Yaskawa INFORM job: FACE.JBI

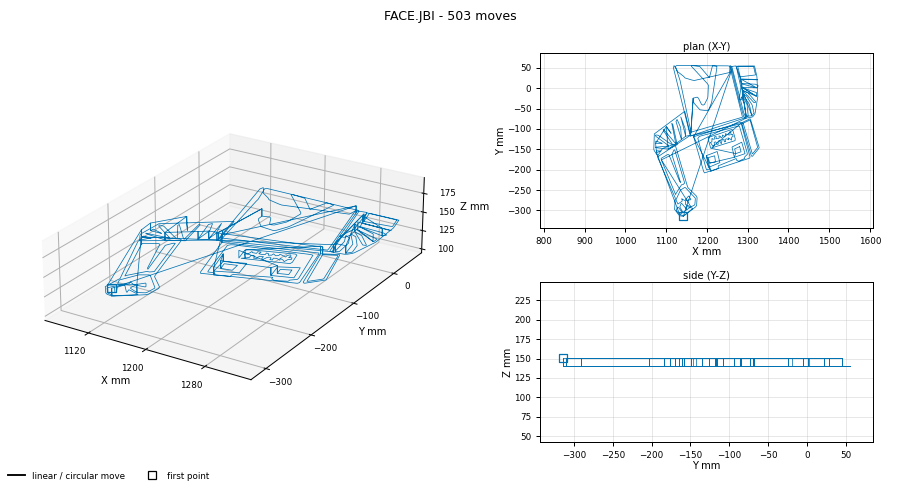
[picture p0: tool path of FACE.JBI, 503 of 503 moves have a stored position in this frame; points joined in program order, loops and branches not executed]
/JOB
//NAME FACE
//POS
///NPOS 503,0,0,0
///TOOL 0
///RECTAN
///RCONF 0,0,0,0,0
C000=1142.216,-314.393,150.400,-168.90,-11.30,-68.01
C001=1142.216,-314.393,140.400,-168.90,-11.30,-68.01
C002=1134.449,-313.129,140.400,-168.90,-11.30,-68.01
C003=1131.072,-310.829,140.400,-168.90,-11.30,-68.01
C004=1123.379,-300.418,140.400,-168.90,-11.30,-68.01
C005=1120.882,-297.547,140.400,-168.90,-11.30,-68.01
C006=1122.133,-274.567,140.400,-168.90,-11.30,-68.01
C007=1122.718,-270.045,140.400,-168.90,-11.30,-68.01
C008=1079.751,-170.531,140.400,-168.90,-11.30,-68.01
C009=1079.155,-166.216,140.400,-168.90,-11.30,-68.01
C010=1089.747,-150.034,140.400,-168.90,-11.30,-68.01
C011=1092.880,-147.217,140.400,-168.90,-11.30,-68.01
C012=1119.146,-137.682,140.400,-168.90,-11.30,-68.01
C013=1122.343,-138.803,140.400,-168.90,-11.30,-68.01
C014=1152.037,-239.693,140.400,-168.90,-11.30,-68.01
C015=1153.633,-243.991,140.400,-168.90,-11.30,-68.01
C016=1174.508,-264.668,140.400,-168.90,-11.30,-68.01
C017=1176.099,-268.887,140.400,-168.90,-11.30,-68.01
C018=1174.919,-287.456,140.400,-168.90,-11.30,-68.01
C019=1172.572,-291.099,140.400,-168.90,-11.30,-68.01
C020=1142.216,-314.393,140.400,-168.90,-11.30,-68.01
C021=1142.216,-314.393,150.400,-168.90,-11.30,-68.01
C022=1261.140,45.571,150.400,-168.90,-11.30,-68.01
C023=1261.140,45.571,140.400,-168.90,-11.30,-68.01
C024=1259.390,51.970,140.400,-168.90,-11.30,-68.01
C025=1260.185,53.171,140.400,-168.90,-11.30,-68.01
C026=1270.179,54.649,140.400,-168.90,-11.30,-68.01
C027=1271.844,54.481,140.400,-168.90,-11.30,-68.01
C028=1284.953,15.522,140.400,-168.90,-11.30,-68.01
C029=1285.567,13.659,140.400,-168.90,-11.30,-68.01
C030=1288.428,-16.125,140.400,-168.90,-11.30,-68.01
C031=1288.496,-18.132,140.400,-168.90,-11.30,-68.01
C032=1286.518,-25.689,140.400,-168.90,-11.30,-68.01
C033=1285.431,-27.217,140.400,-168.90,-11.30,-68.01
C034=1279.741,-28.523,140.400,-168.90,-11.30,-68.01
C035=1278.883,-26.796,140.400,-168.90,-11.30,-68.01
C036=1261.140,45.571,140.400,-168.90,-11.30,-68.01
C037=1261.140,45.571,150.400,-168.90,-11.30,-68.01
C038=1167.569,-118.998,150.400,-168.90,-11.30,-68.01
C039=1167.569,-118.998,140.400,-168.90,-11.30,-68.01
C040=1192.088,-204.021,140.400,-168.90,-11.30,-68.01
C041=1194.246,-207.832,140.400,-168.90,-11.30,-68.01
C042=1304.761,-171.662,140.400,-168.90,-11.30,-68.01
C043=1306.027,-168.728,140.400,-168.90,-11.30,-68.01
C044=1284.671,-87.221,140.400,-168.90,-11.30,-68.01
C045=1282.926,-83.931,140.400,-168.90,-11.30,-68.01
C046=1167.569,-118.998,140.400,-168.90,-11.30,-68.01
C047=1167.569,-118.998,150.400,-168.90,-11.30,-68.01
C048=1210.073,-203.554,150.400,-168.90,-11.30,-68.01
C049=1210.073,-203.554,140.400,-168.90,-11.30,-68.01
C050=1209.248,-199.690,140.400,-168.90,-11.30,-68.01
C051=1206.969,-198.014,140.400,-168.90,-11.30,-68.01
C052=1199.596,-200.286,140.400,-168.90,-11.30,-68.01
C053=1197.924,-196.449,140.400,-168.90,-11.30,-68.01
C054=1179.234,-127.323,140.400,-168.90,-11.30,-68.01
C055=1177.887,-123.066,140.400,-168.90,-11.30,-68.01
C056=1180.126,-119.606,140.400,-168.90,-11.30,-68.01
C057=1183.560,-117.586,140.400,-168.90,-11.30,-68.01
C058=1276.639,-93.033,140.400,-168.90,-11.30,-68.01
C059=1280.079,-93.364,140.400,-168.90,-11.30,-68.01
C060=1298.770,-157.796,140.400,-168.90,-11.30,-68.01
C061=1299.402,-162.315,140.400,-168.90,-11.30,-68.01
C062=1292.772,-168.751,140.400,-168.90,-11.30,-68.01
C063=1292.835,-172.554,140.400,-168.90,-11.30,-68.01
C064=1282.048,-177.222,140.400,-168.90,-11.30,-68.01
C065=1278.602,-179.227,140.400,-168.90,-11.30,-68.01
C066=1273.121,-176.889,140.400,-168.90,-11.30,-68.01
C067=1271.997,-172.516,140.400,-168.90,-11.30,-68.01
C068=1232.551,-188.683,140.400,-168.90,-11.30,-68.01
C069=1228.879,-189.649,140.400,-168.90,-11.30,-68.01
C070=1227.803,-192.650,140.400,-168.90,-11.30,-68.01
C071=1228.391,-196.968,140.400,-168.90,-11.30,-68.01
C072=1210.073,-203.554,140.400,-168.90,-11.30,-68.01
C073=1210.073,-203.554,150.400,-168.90,-11.30,-68.01
C074=1198.888,-165.385,150.400,-168.90,-11.30,-68.01
C075=1198.888,-165.385,140.400,-168.90,-11.30,-68.01
C076=1224.557,-155.662,140.400,-168.90,-11.30,-68.01
C077=1225.399,-155.312,140.400,-168.90,-11.30,-68.01
C078=1231.871,-181.292,140.400,-168.90,-11.30,-68.01
C079=1232.046,-182.567,140.400,-168.90,-11.30,-68.01
C080=1205.150,-193.928,140.400,-168.90,-11.30,-68.01
C081=1204.074,-193.882,140.400,-168.90,-11.30,-68.01
C082=1198.888,-165.385,140.400,-168.90,-11.30,-68.01
C083=1198.888,-165.385,150.400,-168.90,-11.30,-68.01
C084=1207.090,-183.673,150.400,-168.90,-11.30,-68.01
C085=1207.090,-183.673,140.400,-168.90,-11.30,-68.01
C086=1203.439,-170.595,140.400,-168.90,-11.30,-68.01
C087=1203.647,-170.151,140.400,-168.90,-11.30,-68.01
C088=1218.665,-166.291,140.400,-168.90,-11.30,-68.01
C089=1219.146,-165.907,140.400,-168.90,-11.30,-68.01
C090=1221.234,-180.247,140.400,-168.90,-11.30,-68.01
C091=1221.310,-180.935,140.400,-168.90,-11.30,-68.01
C092=1207.090,-183.673,140.400,-168.90,-11.30,-68.01
C093=1207.090,-183.673,150.400,-168.90,-11.30,-68.01
C094=1267.490,-169.400,150.400,-168.90,-11.30,-68.01
C095=1267.490,-169.400,140.400,-168.90,-11.30,-68.01
C096=1261.912,-145.035,140.400,-168.90,-11.30,-68.01
C097=1262.299,-143.982,140.400,-168.90,-11.30,-68.01
C098=1284.598,-132.883,140.400,-168.90,-11.30,-68.01
C099=1285.605,-132.441,140.400,-168.90,-11.30,-68.01
C100=1293.423,-159.373,140.400,-168.90,-11.30,-68.01
C101=1293.680,-160.612,140.400,-168.90,-11.30,-68.01
C102=1267.490,-169.400,140.400,-168.90,-11.30,-68.01
C103=1267.490,-169.400,150.400,-168.90,-11.30,-68.01
C104=1270.846,-160.479,150.400,-168.90,-11.30,-68.01
C105=1270.846,-160.479,140.400,-168.90,-11.30,-68.01
C106=1268.141,-149.422,140.400,-168.90,-11.30,-68.01
C107=1268.264,-148.849,140.400,-168.90,-11.30,-68.01
C108=1280.237,-143.440,140.400,-168.90,-11.30,-68.01
C109=1280.435,-142.889,140.400,-168.90,-11.30,-68.01
C110=1283.781,-155.413,140.400,-168.90,-11.30,-68.01
C111=1283.876,-156.015,140.400,-168.90,-11.30,-68.01
C112=1270.846,-160.479,140.400,-168.90,-11.30,-68.01
C113=1270.846,-160.479,150.400,-168.90,-11.30,-68.01
C114=1209.327,-147.075,150.400,-168.90,-11.30,-68.01
C115=1209.327,-147.075,140.400,-168.90,-11.30,-68.01
C116=1203.871,-126.149,140.400,-168.90,-11.30,-68.01
C117=1203.967,-120.806,140.400,-168.90,-11.30,-68.01
C118=1260.582,-101.433,140.400,-168.90,-11.30,-68.01
C119=1263.748,-103.256,140.400,-168.90,-11.30,-68.01
C120=1269.654,-123.851,140.400,-168.90,-11.30,-68.01
C121=1269.259,-128.629,140.400,-168.90,-11.30,-68.01
C122=1216.586,-144.976,140.400,-168.90,-11.30,-68.01
C123=1212.138,-146.329,140.400,-168.90,-11.30,-68.01
C124=1216.804,-141.922,140.400,-168.90,-11.30,-68.01
C125=1219.065,-139.077,140.400,-168.90,-11.30,-68.01
C126=1217.878,-133.776,140.400,-168.90,-11.30,-68.01
C127=1220.476,-131.362,140.400,-168.90,-11.30,-68.01
C128=1222.990,-132.918,140.400,-168.90,-11.30,-68.01
C129=1224.317,-138.167,140.400,-168.90,-11.30,-68.01
C130=1228.388,-136.987,140.400,-168.90,-11.30,-68.01
C131=1227.101,-132.891,140.400,-168.90,-11.30,-68.01
C132=1228.067,-129.549,140.400,-168.90,-11.30,-68.01
C133=1232.243,-128.372,140.400,-168.90,-11.30,-68.01
C134=1232.971,-133.614,140.400,-168.90,-11.30,-68.01
C135=1235.908,-135.864,140.400,-168.90,-11.30,-68.01
C136=1236.959,-127.903,140.400,-168.90,-11.30,-68.01
C137=1239.103,-125.553,140.400,-168.90,-11.30,-68.01
C138=1241.809,-126.673,140.400,-168.90,-11.30,-68.01
C139=1243.068,-131.537,140.400,-168.90,-11.30,-68.01
C140=1246.286,-130.752,140.400,-168.90,-11.30,-68.01
C141=1244.372,-125.820,140.400,-168.90,-11.30,-68.01
C142=1248.066,-124.071,140.400,-168.90,-11.30,-68.01
C143=1254.018,-126.612,140.400,-168.90,-11.30,-68.01
C144=1251.840,-121.785,140.400,-168.90,-11.30,-68.01
C145=1257.361,-124.563,140.400,-168.90,-11.30,-68.01
C146=1260.353,-127.410,140.400,-168.90,-11.30,-68.01
C147=1261.230,-119.837,140.400,-168.90,-11.30,-68.01
C148=1264.566,-118.155,140.400,-168.90,-11.30,-68.01
C149=1262.828,-113.087,140.400,-168.90,-11.30,-68.01
C150=1258.874,-114.462,140.400,-168.90,-11.30,-68.01
C151=1259.134,-109.099,140.400,-168.90,-11.30,-68.01
C152=1256.703,-106.648,140.400,-168.90,-11.30,-68.01
C153=1254.283,-110.349,140.400,-168.90,-11.30,-68.01
C154=1255.100,-115.131,140.400,-168.90,-11.30,-68.01
C155=1248.357,-112.577,140.400,-168.90,-11.30,-68.01
C156=1245.205,-111.607,140.400,-168.90,-11.30,-68.01
C157=1245.919,-115.773,140.400,-168.90,-11.30,-68.01
C158=1243.087,-118.272,140.400,-168.90,-11.30,-68.01
C159=1240.242,-116.315,140.400,-168.90,-11.30,-68.01
C160=1238.240,-114.840,140.400,-168.90,-11.30,-68.01
C161=1238.162,-119.407,140.400,-168.90,-11.30,-68.01
C162=1234.760,-121.587,140.400,-168.90,-11.30,-68.01
C163=1233.140,-117.823,140.400,-168.90,-11.30,-68.01
C164=1229.650,-117.080,140.400,-168.90,-11.30,-68.01
C165=1230.708,-122.045,140.400,-168.90,-11.30,-68.01
C166=1226.627,-123.850,140.400,-168.90,-11.30,-68.01
C167=1222.963,-123.861,140.400,-168.90,-11.30,-68.01
C168=1222.873,-118.425,140.400,-168.90,-11.30,-68.01
C169=1218.732,-119.333,140.400,-168.90,-11.30,-68.01
C170=1220.063,-124.490,140.400,-168.90,-11.30,-68.01
C171=1214.768,-125.166,140.400,-168.90,-11.30,-68.01
C172=1212.656,-122.721,140.400,-168.90,-11.30,-68.01
C173=1212.363,-131.840,140.400,-168.90,-11.30,-68.01
C174=1208.585,-133.069,140.400,-168.90,-11.30,-68.01
C175=1215.153,-142.336,140.400,-168.90,-11.30,-68.01
C176=1215.153,-142.336,150.400,-168.90,-11.30,-68.01
C177=1285.572,-84.813,150.400,-168.90,-11.30,-68.01
C178=1285.572,-84.813,140.400,-168.90,-11.30,-68.01
C179=1308.142,-163.024,140.400,-168.90,-11.30,-68.01
C180=1308.881,-165.097,140.400,-168.90,-11.30,-68.01
C181=1310.037,-166.717,140.400,-168.90,-11.30,-68.01
C182=1311.890,-167.044,140.400,-168.90,-11.30,-68.01
C183=1327.414,-147.745,140.400,-168.90,-11.30,-68.01
C184=1328.473,-145.985,140.400,-168.90,-11.30,-68.01
C185=1307.240,-76.651,140.400,-168.90,-11.30,-68.01
C186=1306.065,-74.894,140.400,-168.90,-11.30,-68.01
C187=1285.572,-84.813,140.400,-168.90,-11.30,-68.01
C188=1285.572,-84.813,150.400,-168.90,-11.30,-68.01
C189=1289.129,-85.833,150.400,-168.90,-11.30,-68.01
C190=1289.129,-85.833,140.400,-168.90,-11.30,-68.01
C191=1305.172,-78.214,140.400,-168.90,-11.30,-68.01
C192=1306.452,-79.291,140.400,-168.90,-11.30,-68.01
C193=1324.306,-143.586,140.400,-168.90,-11.30,-68.01
C194=1324.428,-145.580,140.400,-168.90,-11.30,-68.01
C195=1312.987,-159.953,140.400,-168.90,-11.30,-68.01
C196=1311.571,-160.939,140.400,-168.90,-11.30,-68.01
C197=1289.129,-85.833,140.400,-168.90,-11.30,-68.01
C198=1289.129,-85.833,150.400,-168.90,-11.30,-68.01
C199=1159.360,-117.208,150.400,-168.90,-11.30,-68.01
C200=1159.360,-117.208,140.400,-168.90,-11.30,-68.01
C201=1118.180,49.460,140.400,-168.90,-11.30,-68.01
C202=1119.497,55.571,140.400,-168.90,-11.30,-68.01
C203=1125.664,46.018,140.400,-168.90,-11.30,-68.01
C204=1128.627,40.362,140.400,-168.90,-11.30,-68.01
C205=1142.318,29.801,140.400,-168.90,-11.30,-68.01
C206=1146.705,25.134,140.400,-168.90,-11.30,-68.01
C207=1163.408,20.106,140.400,-168.90,-11.30,-68.01
C208=1169.188,18.923,140.400,-168.90,-11.30,-68.01
C209=1249.754,37.195,140.400,-168.90,-11.30,-68.01
C210=1255.523,38.485,140.400,-168.90,-11.30,-68.01
C211=1257.363,55.406,140.400,-168.90,-11.30,-68.01
C212=1261.358,52.920,140.400,-168.90,-11.30,-68.01
C213=1290.500,-59.941,140.400,-168.90,-11.30,-68.01
C214=1293.285,-66.126,140.400,-168.90,-11.30,-68.01
C215=1294.241,-72.557,140.400,-168.90,-11.30,-68.01
C216=1159.360,-117.208,140.400,-168.90,-11.30,-68.01
C217=1159.360,-117.208,150.400,-168.90,-11.30,-68.01
C218=1161.224,-107.842,150.400,-168.90,-11.30,-68.01
C219=1161.224,-107.842,140.400,-168.90,-11.30,-68.01
C220=1135.369,12.698,140.400,-168.90,-11.30,-68.01
C221=1134.326,18.823,140.400,-168.90,-11.30,-68.01
C222=1122.945,53.527,140.400,-168.90,-11.30,-68.01
C223=1126.131,55.684,140.400,-168.90,-11.30,-68.01
C224=1251.144,54.899,140.400,-168.90,-11.30,-68.01
C225=1256.222,54.233,140.400,-168.90,-11.30,-68.01
C226=1286.248,-65.099,140.400,-168.90,-11.30,-68.01
C227=1287.500,-71.055,140.400,-168.90,-11.30,-68.01
C228=1161.224,-107.842,140.400,-168.90,-11.30,-68.01
C229=1161.224,-107.842,150.400,-168.90,-11.30,-68.01
C230=1166.451,-24.439,150.400,-168.90,-11.30,-68.01
C231=1166.451,-24.439,140.400,-168.90,-11.30,-68.01
C232=1167.115,-33.389,140.400,-168.90,-11.30,-68.01
C233=1169.138,-37.290,140.400,-168.90,-11.30,-68.01
C234=1180.240,-49.980,140.400,-168.90,-11.30,-68.01
C235=1183.118,-53.016,140.400,-168.90,-11.30,-68.01
C236=1201.565,-55.309,140.400,-168.90,-11.30,-68.01
C237=1204.602,-52.617,140.400,-168.90,-11.30,-68.01
C238=1211.335,-36.119,140.400,-168.90,-11.30,-68.01
C239=1212.336,-31.691,140.400,-168.90,-11.30,-68.01
C240=1224.360,49.148,140.400,-168.90,-11.30,-68.01
C241=1224.666,53.731,140.400,-168.90,-11.30,-68.01
C242=1217.583,54.812,140.400,-168.90,-11.30,-68.01
C243=1213.740,54.836,140.400,-168.90,-11.30,-68.01
C244=1207.453,30.125,140.400,-168.90,-11.30,-68.01
C245=1206.273,25.760,140.400,-168.90,-11.30,-68.01
C246=1185.479,50.031,140.400,-168.90,-11.30,-68.01
C247=1182.760,53.284,140.400,-168.90,-11.30,-68.01
C248=1164.086,55.646,140.400,-168.90,-11.30,-68.01
C249=1162.003,53.955,140.400,-168.90,-11.30,-68.01
C250=1201.673,10.918,140.400,-168.90,-11.30,-68.01
C251=1203.836,7.312,140.400,-168.90,-11.30,-68.01
C252=1202.662,-19.919,140.400,-168.90,-11.30,-68.01
C253=1202.007,-24.366,140.400,-168.90,-11.30,-68.01
C254=1196.121,-36.139,140.400,-168.90,-11.30,-68.01
C255=1194.018,-39.982,140.400,-168.90,-11.30,-68.01
C256=1190.666,-41.447,140.400,-168.90,-11.30,-68.01
C257=1187.074,-39.865,140.400,-168.90,-11.30,-68.01
C258=1179.376,-24.325,140.400,-168.90,-11.30,-68.01
C259=1176.184,-21.874,140.400,-168.90,-11.30,-68.01
C260=1166.451,-24.439,140.400,-168.90,-11.30,-68.01
C261=1166.451,-24.439,150.400,-168.90,-11.30,-68.01
C262=1160.167,-115.279,150.400,-168.90,-11.30,-68.01
C263=1160.167,-115.279,140.400,-168.90,-11.30,-68.01
C264=1082.723,-165.859,140.400,-168.90,-11.30,-68.01
C265=1080.313,-167.741,140.400,-168.90,-11.30,-68.01
C266=1071.067,-153.243,140.400,-168.90,-11.30,-68.01
C267=1069.888,-150.113,140.400,-168.90,-11.30,-68.01
C268=1071.053,-115.578,140.400,-168.90,-11.30,-68.01
C269=1071.159,-112.110,140.400,-168.90,-11.30,-68.01
C270=1143.371,-58.422,140.400,-168.90,-11.30,-68.01
C271=1145.966,-56.870,140.400,-168.90,-11.30,-68.01
C272=1160.167,-115.279,140.400,-168.90,-11.30,-68.01
C273=1160.167,-115.279,150.400,-168.90,-11.30,-68.01
C274=1148.039,-117.802,150.400,-168.90,-11.30,-68.01
C275=1148.039,-117.802,140.400,-168.90,-11.30,-68.01
C276=1136.303,-71.473,140.400,-168.90,-11.30,-68.01
C277=1136.182,-70.430,140.400,-168.90,-11.30,-68.01
C278=1146.348,-97.663,140.400,-168.90,-11.30,-68.01
C279=1146.644,-98.652,140.400,-168.90,-11.30,-68.01
C280=1148.039,-117.802,140.400,-168.90,-11.30,-68.01
C281=1148.039,-117.802,150.400,-168.90,-11.30,-68.01
C282=1137.758,-126.003,150.400,-168.90,-11.30,-68.01
C283=1137.758,-126.003,140.400,-168.90,-11.30,-68.01
C284=1124.533,-82.682,140.400,-168.90,-11.30,-68.01
C285=1124.399,-81.618,140.400,-168.90,-11.30,-68.01
C286=1126.531,-77.034,140.400,-168.90,-11.30,-68.01
C287=1127.330,-77.266,140.400,-168.90,-11.30,-68.01
C288=1135.422,-95.367,140.400,-168.90,-11.30,-68.01
C289=1135.740,-96.382,140.400,-168.90,-11.30,-68.01
C290=1137.758,-126.003,140.400,-168.90,-11.30,-68.01
C291=1137.758,-126.003,150.400,-168.90,-11.30,-68.01
C292=1105.212,-149.417,150.400,-168.90,-11.30,-68.01
C293=1105.212,-149.417,140.400,-168.90,-11.30,-68.01
C294=1077.154,-146.213,140.400,-168.90,-11.30,-68.01
C295=1073.706,-144.770,140.400,-168.90,-11.30,-68.01
C296=1104.977,-142.002,140.400,-168.90,-11.30,-68.01
C297=1105.747,-140.590,140.400,-168.90,-11.30,-68.01
C298=1075.163,-118.410,140.400,-168.90,-11.30,-68.01
C299=1073.568,-115.166,140.400,-168.90,-11.30,-68.01
C300=1077.111,-114.843,140.400,-168.90,-11.30,-68.01
C301=1080.719,-115.437,140.400,-168.90,-11.30,-68.01
C302=1112.033,-137.127,140.400,-168.90,-11.30,-68.01
C303=1115.630,-137.905,140.400,-168.90,-11.30,-68.01
C304=1093.632,-103.960,140.400,-168.90,-11.30,-68.01
C305=1093.807,-100.838,140.400,-168.90,-11.30,-68.01
C306=1121.935,-134.174,140.400,-168.90,-11.30,-68.01
C307=1123.699,-135.364,140.400,-168.90,-11.30,-68.01
C308=1113.941,-86.034,140.400,-168.90,-11.30,-68.01
C309=1116.389,-88.667,140.400,-168.90,-11.30,-68.01
C310=1126.572,-134.597,140.400,-168.90,-11.30,-68.01
C311=1127.246,-138.494,140.400,-168.90,-11.30,-68.01
C312=1105.212,-149.417,140.400,-168.90,-11.30,-68.01
C313=1105.212,-149.417,150.400,-168.90,-11.30,-68.01
C314=1100.585,-94.148,150.400,-168.90,-11.30,-68.01
C315=1100.585,-94.148,140.400,-168.90,-11.30,-68.01
C316=1112.231,-110.790,140.400,-168.90,-11.30,-68.01
C317=1112.510,-110.690,140.400,-168.90,-11.30,-68.01
C318=1100.585,-94.148,140.400,-168.90,-11.30,-68.01
C319=1100.585,-94.148,150.400,-168.90,-11.30,-68.01
C320=1074.221,-135.149,150.400,-168.90,-11.30,-68.01
C321=1074.221,-135.149,140.400,-168.90,-11.30,-68.01
C322=1074.783,-129.726,140.400,-168.90,-11.30,-68.01
C323=1075.213,-129.714,140.400,-168.90,-11.30,-68.01
C324=1090.419,-134.983,140.400,-168.90,-11.30,-68.01
C325=1090.426,-135.339,140.400,-168.90,-11.30,-68.01
C326=1074.221,-135.149,140.400,-168.90,-11.30,-68.01
C327=1074.221,-135.149,150.400,-168.90,-11.30,-68.01
C328=1076.594,-158.173,150.400,-168.90,-11.30,-68.01
C329=1076.594,-158.173,140.400,-168.90,-11.30,-68.01
C330=1076.551,-153.713,140.400,-168.90,-11.30,-68.01
C331=1076.844,-153.586,140.400,-168.90,-11.30,-68.01
C332=1087.342,-153.880,140.400,-168.90,-11.30,-68.01
C333=1087.625,-154.033,140.400,-168.90,-11.30,-68.01
C334=1076.594,-158.173,140.400,-168.90,-11.30,-68.01
C335=1076.594,-158.173,150.400,-168.90,-11.30,-68.01
C336=1133.276,-309.876,150.400,-168.90,-11.30,-68.01
C337=1133.276,-309.876,140.400,-168.90,-11.30,-68.01
C338=1125.215,-299.949,140.400,-168.90,-11.30,-68.01
C339=1124.975,-298.206,140.400,-168.90,-11.30,-68.01
C340=1128.684,-291.471,140.400,-168.90,-11.30,-68.01
C341=1130.078,-292.062,140.400,-168.90,-11.30,-68.01
C342=1139.644,-304.606,140.400,-168.90,-11.30,-68.01
C343=1140.719,-303.448,140.400,-168.90,-11.30,-68.01
C344=1134.335,-292.498,140.400,-168.90,-11.30,-68.01
C345=1133.868,-290.818,140.400,-168.90,-11.30,-68.01
C346=1136.688,-283.104,140.400,-168.90,-11.30,-68.01
C347=1138.027,-282.345,140.400,-168.90,-11.30,-68.01
C348=1149.695,-296.072,140.400,-168.90,-11.30,-68.01
C349=1151.057,-296.763,140.400,-168.90,-11.30,-68.01
C350=1148.945,-290.513,140.400,-168.90,-11.30,-68.01
C351=1149.627,-289.966,140.400,-168.90,-11.30,-68.01
C352=1164.746,-294.464,140.400,-168.90,-11.30,-68.01
C353=1164.800,-295.669,140.400,-168.90,-11.30,-68.01
C354=1144.562,-312.032,140.400,-168.90,-11.30,-68.01
C355=1143.228,-312.778,140.400,-168.90,-11.30,-68.01
C356=1133.276,-309.876,140.400,-168.90,-11.30,-68.01
C357=1133.276,-309.876,150.400,-168.90,-11.30,-68.01
C358=1161.138,-291.143,150.400,-168.90,-11.30,-68.01
C359=1161.138,-291.143,140.400,-168.90,-11.30,-68.01
C360=1148.390,-285.735,140.400,-168.90,-11.30,-68.01
C361=1147.310,-283.863,140.400,-168.90,-11.30,-68.01
C362=1148.084,-277.199,140.400,-168.90,-11.30,-68.01
C363=1149.036,-275.186,140.400,-168.90,-11.30,-68.01
C364=1160.089,-273.689,140.400,-168.90,-11.30,-68.01
C365=1160.999,-272.733,140.400,-168.90,-11.30,-68.01
C366=1156.562,-265.916,140.400,-168.90,-11.30,-68.01
C367=1154.985,-264.545,140.400,-168.90,-11.30,-68.01
C368=1147.437,-274.225,140.400,-168.90,-11.30,-68.01
C369=1145.760,-275.419,140.400,-168.90,-11.30,-68.01
C370=1139.277,-271.868,140.400,-168.90,-11.30,-68.01
C371=1138.549,-271.094,140.400,-168.90,-11.30,-68.01
C372=1139.562,-275.582,140.400,-168.90,-11.30,-68.01
C373=1139.050,-277.429,140.400,-168.90,-11.30,-68.01
C374=1130.830,-283.209,140.400,-168.90,-11.30,-68.01
C375=1129.083,-284.155,140.400,-168.90,-11.30,-68.01
C376=1124.790,-275.255,140.400,-168.90,-11.30,-68.01
C377=1124.572,-272.934,140.400,-168.90,-11.30,-68.01
C378=1134.404,-251.704,140.400,-168.90,-11.30,-68.01
C379=1135.483,-249.778,140.400,-168.90,-11.30,-68.01
C380=1145.723,-243.540,140.400,-168.90,-11.30,-68.01
C381=1147.612,-244.026,140.400,-168.90,-11.30,-68.01
C382=1170.857,-268.775,140.400,-168.90,-11.30,-68.01
C383=1171.791,-270.708,140.400,-168.90,-11.30,-68.01
C384=1170.732,-284.556,140.400,-168.90,-11.30,-68.01
C385=1169.865,-286.593,140.400,-168.90,-11.30,-68.01
C386=1161.138,-291.143,140.400,-168.90,-11.30,-68.01
C387=1161.138,-291.143,150.400,-168.90,-11.30,-68.01
C388=1088.457,-175.834,150.400,-168.90,-11.30,-68.01
C389=1088.457,-175.834,140.400,-168.90,-11.30,-68.01
C390=1087.829,-172.141,140.400,-168.90,-11.30,-68.01
C391=1103.994,-162.627,140.400,-168.90,-11.30,-68.01
C392=1106.994,-163.095,140.400,-168.90,-11.30,-68.01
C393=1133.317,-228.730,140.400,-168.90,-11.30,-68.01
C394=1135.527,-231.148,140.400,-168.90,-11.30,-68.01
C395=1115.703,-166.642,140.400,-168.90,-11.30,-68.01
C396=1114.258,-162.665,140.400,-168.90,-11.30,-68.01
C397=1118.918,-152.318,140.400,-168.90,-11.30,-68.01
C398=1121.287,-151.255,140.400,-168.90,-11.30,-68.01
C399=1144.414,-228.514,140.400,-168.90,-11.30,-68.01
C400=1145.614,-232.605,140.400,-168.90,-11.30,-68.01
C401=1141.572,-236.501,140.400,-168.90,-11.30,-68.01
C402=1137.999,-236.874,140.400,-168.90,-11.30,-68.01
C403=1124.795,-257.451,140.400,-168.90,-11.30,-68.01
C404=1123.339,-261.032,140.400,-168.90,-11.30,-68.01
C405=1088.457,-175.834,140.400,-168.90,-11.30,-68.01
C406=1088.457,-175.834,150.400,-168.90,-11.30,-68.01
C407=1296.525,-73.313,150.400,-168.90,-11.30,-68.01
C408=1296.525,-73.313,140.400,-168.90,-11.30,-68.01
C409=1293.606,-73.138,140.400,-168.90,-11.30,-68.01
C410=1291.082,-71.805,140.400,-168.90,-11.30,-68.01
C411=1280.170,-32.310,140.400,-168.90,-11.30,-68.01
C412=1279.207,-29.008,140.400,-168.90,-11.30,-68.01
C413=1283.463,0.131,140.400,-168.90,-11.30,-68.01
C414=1283.196,3.554,140.400,-168.90,-11.30,-68.01
C415=1272.952,50.537,140.400,-168.90,-11.30,-68.01
C416=1271.757,53.653,140.400,-168.90,-11.30,-68.01
C417=1314.201,53.617,140.400,-168.90,-11.30,-68.01
C418=1316.956,54.676,140.400,-168.90,-11.30,-68.01
C419=1322.261,31.831,140.400,-168.90,-11.30,-68.01
C420=1322.864,28.410,140.400,-168.90,-11.30,-68.01
C421=1324.803,-16.851,140.400,-168.90,-11.30,-68.01
C422=1325.133,-20.319,140.400,-168.90,-11.30,-68.01
C423=1318.520,-60.795,140.400,-168.90,-11.30,-68.01
C424=1317.282,-63.906,140.400,-168.90,-11.30,-68.01
C425=1313.432,-69.039,140.400,-168.90,-11.30,-68.01
C426=1310.926,-70.831,140.400,-168.90,-11.30,-68.01
C427=1296.525,-73.313,140.400,-168.90,-11.30,-68.01
C428=1296.525,-73.313,150.400,-168.90,-11.30,-68.01
C429=1281.984,28.048,150.400,-168.90,-11.30,-68.01
C430=1281.984,28.048,140.400,-168.90,-11.30,-68.01
C431=1275.872,52.915,140.400,-168.90,-11.30,-68.01
C432=1275.614,54.336,140.400,-168.90,-11.30,-68.01
C433=1313.156,54.431,140.400,-168.90,-11.30,-68.01
C434=1314.362,54.642,140.400,-168.90,-11.30,-68.01
C435=1319.414,34.043,140.400,-168.90,-11.30,-68.01
C436=1319.504,32.586,140.400,-168.90,-11.30,-68.01
C437=1281.984,28.048,140.400,-168.90,-11.30,-68.01
C438=1281.984,28.048,150.400,-168.90,-11.30,-68.01
C439=1296.944,-69.935,150.400,-168.90,-11.30,-68.01
C440=1296.944,-69.935,140.400,-168.90,-11.30,-68.01
C441=1292.095,-39.148,140.400,-168.90,-11.30,-68.01
C442=1291.969,-37.983,140.400,-168.90,-11.30,-68.01
C443=1284.970,-22.514,140.400,-168.90,-11.30,-68.01
C444=1284.827,-21.356,140.400,-168.90,-11.30,-68.01
C445=1291.584,-25.466,140.400,-168.90,-11.30,-68.01
C446=1292.304,-26.269,140.400,-168.90,-11.30,-68.01
C447=1298.477,-39.585,140.400,-168.90,-11.30,-68.01
C448=1298.775,-40.709,140.400,-168.90,-11.30,-68.01
C449=1301.432,-66.352,140.400,-168.90,-11.30,-68.01
C450=1301.360,-67.528,140.400,-168.90,-11.30,-68.01
C451=1296.944,-69.042,140.400,-168.90,-11.30,-68.01
C452=1296.944,-69.042,150.400,-168.90,-11.30,-68.01
C453=1310.460,-67.570,150.400,-168.90,-11.30,-68.01
C454=1310.460,-67.570,140.400,-168.90,-11.30,-68.01
C455=1304.638,-40.138,140.400,-168.90,-11.30,-68.01
C456=1304.113,-38.903,140.400,-168.90,-11.30,-68.01
C457=1287.782,-14.830,140.400,-168.90,-11.30,-68.01
C458=1287.274,-13.960,140.400,-168.90,-11.30,-68.01
C459=1296.353,-18.213,140.400,-168.90,-11.30,-68.01
C460=1297.212,-19.145,140.400,-168.90,-11.30,-68.01
C461=1310.544,-39.788,140.400,-168.90,-11.30,-68.01
C462=1311.110,-40.997,140.400,-168.90,-11.30,-68.01
C463=1315.442,-59.501,140.400,-168.90,-11.30,-68.01
C464=1315.456,-60.887,140.400,-168.90,-11.30,-68.01
C465=1310.460,-67.570,140.400,-168.90,-11.30,-68.01
C466=1310.460,-67.570,150.400,-168.90,-11.30,-68.01
C467=1288.083,-5.494,150.400,-168.90,-11.30,-68.01
C468=1288.083,-5.494,140.400,-168.90,-11.30,-68.01
C469=1315.192,-34.813,140.400,-168.90,-11.30,-68.01
C470=1315.838,-35.484,140.400,-168.90,-11.30,-68.01
C471=1319.767,-34.464,140.400,-168.90,-11.30,-68.01
C472=1319.904,-33.457,140.400,-168.90,-11.30,-68.01
C473=1301.932,-12.205,140.400,-168.90,-11.30,-68.01
C474=1301.244,-11.597,140.400,-168.90,-11.30,-68.01
C475=1288.083,-5.494,140.400,-168.90,-11.30,-68.01
C476=1288.083,-5.494,150.400,-168.90,-11.30,-68.01
C477=1321.365,-19.733,150.400,-168.90,-11.30,-68.01
C478=1321.365,-19.733,140.400,-168.90,-11.30,-68.01
C479=1286.820,1.268,140.400,-168.90,-11.30,-68.01
C480=1286.080,1.688,140.400,-168.90,-11.30,-68.01
C481=1321.239,-10.300,140.400,-168.90,-11.30,-68.01
C482=1322.050,-10.808,140.400,-168.90,-11.30,-68.01
C483=1322.296,-19.290,140.400,-168.90,-11.30,-68.01
C484=1321.466,-19.720,140.400,-168.90,-11.30,-68.01
C485=1287.717,2.234,140.400,-168.90,-11.30,-68.01
C486=1287.717,2.234,150.400,-168.90,-11.30,-68.01
C487=1322.484,0.985,150.400,-168.90,-11.30,-68.01
C488=1322.484,0.985,140.400,-168.90,-11.30,-68.01
C489=1325.808,5.259,140.400,-168.90,-11.30,-68.01
C490=1325.747,6.338,140.400,-168.90,-11.30,-68.01
C491=1320.212,9.507,140.400,-168.90,-11.30,-68.01
C492=1319.342,9.813,140.400,-168.90,-11.30,-68.01
C493=1285.382,11.564,140.400,-168.90,-11.30,-68.01
C494=1284.794,10.815,140.400,-168.90,-11.30,-68.01
C495=1322.484,0.985,140.400,-168.90,-11.30,-68.01
C496=1322.484,0.985,150.400,-168.90,-11.30,-68.01
C497=1284.268,21.948,150.400,-168.90,-11.30,-68.01
C498=1284.268,21.948,140.400,-168.90,-11.30,-68.01
C499=1324.387,20.638,140.400,-168.90,-11.30,-68.01
C500=1323.854,21.444,140.400,-168.90,-11.30,-68.01
C501=1283.522,22.617,140.400,-168.90,-11.30,-68.01
C502=1283.522,22.617,150.400,-168.90,-11.30,-68.01
//INST
///DATE 2014/11/05 02:53
///ATTR 0,0,0,0,0,0,0,0,0,0,0,0,1,1,0,0
///FRAME BASE
NOP
*1
MOVL C000 V=200.0 CONT
PAUSE
MOVL C001 V=50.0 CONT
MOVL C002 V=50.0 CONT
MOVL C003 V=50.0 CONT
MOVL C004 V=50.0 CONT
MOVL C005 V=50.0 CONT
MOVL C006 V=50.0 CONT
MOVL C007 V=50.0 CONT
MOVL C008 V=50.0 CONT
MOVL C009 V=50.0 CONT
MOVL C010 V=50.0 CONT
MOVL C011 V=50.0 CONT
MOVL C012 V=50.0 CONT
MOVL C013 V=50.0 CONT
MOVL C014 V=50.0 CONT
MOVL C015 V=50.0 CONT
MOVL C016 V=50.0 CONT
MOVL C017 V=50.0 CONT
MOVL C018 V=50.0 CONT
MOVL C019 V=50.0 CONT
MOVL C020 V=50.0 CONT
MOVL C021 V=200.0 CONT
MOVL C022 V=200.0 CONT
MOVL C023 V=50.0 CONT
MOVL C024 V=50.0 CONT
MOVL C025 V=50.0 CONT
MOVL C026 V=50.0 CONT
MOVL C027 V=50.0 CONT
MOVL C028 V=50.0 CONT
MOVL C029 V=50.0 CONT
MOVL C030 V=50.0 CONT
MOVL C031 V=50.0 CONT
MOVL C032 V=50.0 CONT
MOVL C033 V=50.0 CONT
MOVL C034 V=50.0 CONT
MOVL C035 V=50.0 CONT
MOVL C036 V=50.0 CONT
MOVL C037 V=200.0 CONT
MOVL C038 V=200.0 CONT
MOVL C039 V=50.0 CONT
MOVL C040 V=50.0 CONT
MOVL C041 V=50.0 CONT
MOVL C042 V=50.0 CONT
MOVL C043 V=50.0 CONT
MOVL C044 V=50.0 CONT
MOVL C045 V=50.0 CONT
MOVL C046 V=50.0 CONT
MOVL C047 V=200.0 CONT
MOVL C048 V=200.0 CONT
MOVL C049 V=50.0 CONT
MOVL C050 V=50.0 CONT
MOVL C051 V=50.0 CONT
MOVL C052 V=50.0 CONT
MOVL C053 V=50.0 CONT
MOVL C054 V=50.0 CONT
MOVL C055 V=50.0 CONT
MOVL C056 V=50.0 CONT
MOVL C057 V=50.0 CONT
MOVL C058 V=50.0 CONT
MOVL C059 V=50.0 CONT
MOVL C060 V=50.0 CONT
MOVL C061 V=50.0 CONT
MOVL C062 V=50.0 CONT
MOVL C063 V=50.0 CONT
MOVL C064 V=50.0 CONT
MOVL C065 V=50.0 CONT
MOVL C066 V=50.0 CONT
MOVL C067 V=50.0 CONT
MOVL C068 V=50.0 CONT
MOVL C069 V=50.0 CONT
MOVL C070 V=50.0 CONT
MOVL C071 V=50.0 CONT
MOVL C072 V=50.0 CONT
MOVL C073 V=200.0 CONT
MOVL C074 V=200.0 CONT
MOVL C075 V=50.0 CONT
MOVL C076 V=50.0 CONT
MOVL C077 V=50.0 CONT
MOVL C078 V=50.0 CONT
MOVL C079 V=50.0 CONT
MOVL C080 V=50.0 CONT
MOVL C081 V=50.0 CONT
MOVL C082 V=50.0 CONT
MOVL C083 V=200.0 CONT
MOVL C084 V=200.0 CONT
MOVL C085 V=50.0 CONT
MOVL C086 V=50.0 CONT
MOVL C087 V=50.0 CONT
MOVL C088 V=50.0 CONT
MOVL C089 V=50.0 CONT
MOVL C090 V=50.0 CONT
MOVL C091 V=50.0 CONT
MOVL C092 V=50.0 CONT
MOVL C093 V=200.0 CONT
MOVL C094 V=200.0 CONT
MOVL C095 V=50.0 CONT
MOVL C096 V=50.0 CONT
MOVL C097 V=50.0 CONT
MOVL C098 V=50.0 CONT
MOVL C099 V=50.0 CONT
MOVL C100 V=50.0 CONT
MOVL C101 V=50.0 CONT
MOVL C102 V=50.0 CONT
MOVL C103 V=200.0 CONT
MOVL C104 V=200.0 CONT
MOVL C105 V=50.0 CONT
MOVL C106 V=50.0 CONT
MOVL C107 V=50.0 CONT
MOVL C108 V=50.0 CONT
MOVL C109 V=50.0 CONT
MOVL C110 V=50.0 CONT
MOVL C111 V=50.0 CONT
MOVL C112 V=50.0 CONT
MOVL C113 V=200.0 CONT
MOVL C114 V=200.0 CONT
MOVL C115 V=50.0 CONT
MOVL C116 V=50.0 CONT
MOVL C117 V=50.0 CONT
MOVL C118 V=50.0 CONT
MOVL C119 V=50.0 CONT
MOVL C120 V=50.0 CONT
MOVL C121 V=50.0 CONT
MOVL C122 V=50.0 CONT
MOVL C123 V=50.0 CONT
MOVL C124 V=50.0 CONT
MOVL C125 V=50.0 CONT
MOVL C126 V=50.0 CONT
MOVL C127 V=50.0 CONT
MOVL C128 V=50.0 CONT
MOVL C129 V=50.0 CONT
MOVL C130 V=50.0 CONT
MOVL C131 V=50.0 CONT
MOVL C132 V=50.0 CONT
MOVL C133 V=50.0 CONT
MOVL C134 V=50.0 CONT
MOVL C135 V=50.0 CONT
MOVL C136 V=50.0 CONT
MOVL C137 V=50.0 CONT
MOVL C138 V=50.0 CONT
MOVL C139 V=50.0 CONT
MOVL C140 V=50.0 CONT
MOVL C141 V=50.0 CONT
MOVL C142 V=50.0 CONT
MOVL C143 V=50.0 CONT
MOVL C144 V=50.0 CONT
MOVL C145 V=50.0 CONT
MOVL C146 V=50.0 CONT
MOVL C147 V=50.0 CONT
MOVL C148 V=50.0 CONT
MOVL C149 V=50.0 CONT
MOVL C150 V=50.0 CONT
MOVL C151 V=50.0 CONT
MOVL C152 V=50.0 CONT
MOVL C153 V=50.0 CONT
MOVL C154 V=50.0 CONT
MOVL C155 V=50.0 CONT
MOVL C156 V=50.0 CONT
MOVL C157 V=50.0 CONT
MOVL C158 V=50.0 CONT
MOVL C159 V=50.0 CONT
MOVL C160 V=50.0 CONT
MOVL C161 V=50.0 CONT
MOVL C162 V=50.0 CONT
MOVL C163 V=50.0 CONT
MOVL C164 V=50.0 CONT
MOVL C165 V=50.0 CONT
MOVL C166 V=50.0 CONT
MOVL C167 V=50.0 CONT
MOVL C168 V=50.0 CONT
MOVL C169 V=50.0 CONT
MOVL C170 V=50.0 CONT
MOVL C171 V=50.0 CONT
MOVL C172 V=50.0 CONT
MOVL C173 V=50.0 CONT
MOVL C174 V=50.0 CONT
MOVL C175 V=50.0 CONT
MOVL C176 V=200.0 CONT
MOVL C177 V=200.0 CONT
MOVL C178 V=50.0 CONT
MOVL C179 V=50.0 CONT
MOVL C180 V=50.0 CONT
MOVL C181 V=50.0 CONT
MOVL C182 V=50.0 CONT
MOVL C183 V=50.0 CONT
MOVL C184 V=50.0 CONT
MOVL C185 V=50.0 CONT
MOVL C186 V=50.0 CONT
MOVL C187 V=50.0 CONT
MOVL C188 V=200.0 CONT
MOVL C189 V=200.0 CONT
MOVL C190 V=50.0 CONT
MOVL C191 V=50.0 CONT
MOVL C192 V=50.0 CONT
MOVL C193 V=50.0 CONT
MOVL C194 V=50.0 CONT
MOVL C195 V=50.0 CONT
MOVL C196 V=50.0 CONT
MOVL C197 V=50.0 CONT
MOVL C198 V=200.0 CONT
MOVL C199 V=200.0 CONT
MOVL C200 V=50.0 CONT
MOVL C201 V=50.0 CONT
MOVL C202 V=50.0 CONT
MOVL C203 V=50.0 CONT
MOVL C204 V=50.0 CONT
MOVL C205 V=50.0 CONT
MOVL C206 V=50.0 CONT
MOVL C207 V=50.0 CONT
MOVL C208 V=50.0 CONT
MOVL C209 V=50.0 CONT
MOVL C210 V=50.0 CONT
MOVL C211 V=50.0 CONT
MOVL C212 V=50.0 CONT
MOVL C213 V=50.0 CONT
MOVL C214 V=50.0 CONT
MOVL C215 V=50.0 CONT
MOVL C216 V=50.0 CONT
MOVL C217 V=200.0 CONT
MOVL C218 V=200.0 CONT
MOVL C219 V=50.0 CONT
MOVL C220 V=50.0 CONT
MOVL C221 V=50.0 CONT
MOVL C222 V=50.0 CONT
MOVL C223 V=50.0 CONT
MOVL C224 V=50.0 CONT
MOVL C225 V=50.0 CONT
MOVL C226 V=50.0 CONT
MOVL C227 V=50.0 CONT
MOVL C228 V=50.0 CONT
MOVL C229 V=200.0 CONT
MOVL C230 V=200.0 CONT
MOVL C231 V=50.0 CONT
MOVL C232 V=50.0 CONT
MOVL C233 V=50.0 CONT
MOVL C234 V=50.0 CONT
MOVL C235 V=50.0 CONT
MOVL C236 V=50.0 CONT
MOVL C237 V=50.0 CONT
MOVL C238 V=50.0 CONT
MOVL C239 V=50.0 CONT
MOVL C240 V=50.0 CONT
MOVL C241 V=50.0 CONT
MOVL C242 V=50.0 CONT
MOVL C243 V=50.0 CONT
MOVL C244 V=50.0 CONT
MOVL C245 V=50.0 CONT
MOVL C246 V=50.0 CONT
MOVL C247 V=50.0 CONT
MOVL C248 V=50.0 CONT
MOVL C249 V=50.0 CONT
MOVL C250 V=50.0 CONT
MOVL C251 V=50.0 CONT
MOVL C252 V=50.0 CONT
MOVL C253 V=50.0 CONT
MOVL C254 V=50.0 CONT
MOVL C255 V=50.0 CONT
MOVL C256 V=50.0 CONT
MOVL C257 V=50.0 CONT
MOVL C258 V=50.0 CONT
MOVL C259 V=50.0 CONT
MOVL C260 V=50.0 CONT
MOVL C261 V=200.0 CONT
MOVL C262 V=200.0 CONT
MOVL C263 V=50.0 CONT
MOVL C264 V=50.0 CONT
MOVL C265 V=50.0 CONT
MOVL C266 V=50.0 CONT
MOVL C267 V=50.0 CONT
MOVL C268 V=50.0 CONT
MOVL C269 V=50.0 CONT
MOVL C270 V=50.0 CONT
MOVL C271 V=50.0 CONT
MOVL C272 V=50.0 CONT
MOVL C273 V=200.0 CONT
MOVL C274 V=200.0 CONT
MOVL C275 V=50.0 CONT
MOVL C276 V=50.0 CONT
MOVL C277 V=50.0 CONT
MOVL C278 V=50.0 CONT
MOVL C279 V=50.0 CONT
MOVL C280 V=50.0 CONT
MOVL C281 V=200.0 CONT
MOVL C282 V=200.0 CONT
MOVL C283 V=50.0 CONT
MOVL C284 V=50.0 CONT
MOVL C285 V=50.0 CONT
MOVL C286 V=50.0 CONT
MOVL C287 V=50.0 CONT
MOVL C288 V=50.0 CONT
MOVL C289 V=50.0 CONT
MOVL C290 V=50.0 CONT
MOVL C291 V=200.0 CONT
MOVL C292 V=200.0 CONT
MOVL C293 V=50.0 CONT
MOVL C294 V=50.0 CONT
MOVL C295 V=50.0 CONT
MOVL C296 V=50.0 CONT
MOVL C297 V=50.0 CONT
MOVL C298 V=50.0 CONT
MOVL C299 V=50.0 CONT
MOVL C300 V=50.0 CONT
MOVL C301 V=50.0 CONT
MOVL C302 V=50.0 CONT
MOVL C303 V=50.0 CONT
MOVL C304 V=50.0 CONT
MOVL C305 V=50.0 CONT
MOVL C306 V=50.0 CONT
MOVL C307 V=50.0 CONT
MOVL C308 V=50.0 CONT
MOVL C309 V=50.0 CONT
MOVL C310 V=50.0 CONT
MOVL C311 V=50.0 CONT
MOVL C312 V=50.0 CONT
MOVL C313 V=200.0 CONT
MOVL C314 V=200.0 CONT
MOVL C315 V=50.0 CONT
MOVL C316 V=50.0 CONT
MOVL C317 V=50.0 CONT
MOVL C318 V=50.0 CONT
MOVL C319 V=200.0 CONT
MOVL C320 V=200.0 CONT
MOVL C321 V=50.0 CONT
MOVL C322 V=50.0 CONT
MOVL C323 V=50.0 CONT
MOVL C324 V=50.0 CONT
MOVL C325 V=50.0 CONT
MOVL C326 V=50.0 CONT
MOVL C327 V=200.0 CONT
MOVL C328 V=200.0 CONT
MOVL C329 V=50.0 CONT
MOVL C330 V=50.0 CONT
MOVL C331 V=50.0 CONT
MOVL C332 V=50.0 CONT
MOVL C333 V=50.0 CONT
MOVL C334 V=50.0 CONT
MOVL C335 V=200.0 CONT
MOVL C336 V=200.0 CONT
MOVL C337 V=50.0 CONT
MOVL C338 V=50.0 CONT
MOVL C339 V=50.0 CONT
MOVL C340 V=50.0 CONT
MOVL C341 V=50.0 CONT
MOVL C342 V=50.0 CONT
MOVL C343 V=50.0 CONT
MOVL C344 V=50.0 CONT
MOVL C345 V=50.0 CONT
MOVL C346 V=50.0 CONT
MOVL C347 V=50.0 CONT
MOVL C348 V=50.0 CONT
MOVL C349 V=50.0 CONT
MOVL C350 V=50.0 CONT
MOVL C351 V=50.0 CONT
MOVL C352 V=50.0 CONT
MOVL C353 V=50.0 CONT
MOVL C354 V=50.0 CONT
MOVL C355 V=50.0 CONT
MOVL C356 V=50.0 CONT
MOVL C357 V=200.0 CONT
MOVL C358 V=200.0 CONT
MOVL C359 V=50.0 CONT
MOVL C360 V=50.0 CONT
MOVL C361 V=50.0 CONT
MOVL C362 V=50.0 CONT
MOVL C363 V=50.0 CONT
MOVL C364 V=50.0 CONT
MOVL C365 V=50.0 CONT
MOVL C366 V=50.0 CONT
MOVL C367 V=50.0 CONT
MOVL C368 V=50.0 CONT
MOVL C369 V=50.0 CONT
MOVL C370 V=50.0 CONT
MOVL C371 V=50.0 CONT
MOVL C372 V=50.0 CONT
MOVL C373 V=50.0 CONT
MOVL C374 V=50.0 CONT
MOVL C375 V=50.0 CONT
MOVL C376 V=50.0 CONT
MOVL C377 V=50.0 CONT
MOVL C378 V=50.0 CONT
MOVL C379 V=50.0 CONT
MOVL C380 V=50.0 CONT
MOVL C381 V=50.0 CONT
MOVL C382 V=50.0 CONT
MOVL C383 V=50.0 CONT
MOVL C384 V=50.0 CONT
MOVL C385 V=50.0 CONT
MOVL C386 V=50.0 CONT
MOVL C387 V=200.0 CONT
MOVL C388 V=200.0 CONT
MOVL C389 V=50.0 CONT
MOVL C390 V=50.0 CONT
MOVL C391 V=50.0 CONT
MOVL C392 V=50.0 CONT
MOVL C393 V=50.0 CONT
MOVL C394 V=50.0 CONT
MOVL C395 V=50.0 CONT
MOVL C396 V=50.0 CONT
MOVL C397 V=50.0 CONT
MOVL C398 V=50.0 CONT
MOVL C399 V=50.0 CONT
MOVL C400 V=50.0 CONT
MOVL C401 V=50.0 CONT
MOVL C402 V=50.0 CONT
MOVL C403 V=50.0 CONT
MOVL C404 V=50.0 CONT
MOVL C405 V=50.0 CONT
MOVL C406 V=200.0 CONT
MOVL C407 V=200.0 CONT
MOVL C408 V=50.0 CONT
MOVL C409 V=50.0 CONT
MOVL C410 V=50.0 CONT
MOVL C411 V=50.0 CONT
MOVL C412 V=50.0 CONT
MOVL C413 V=50.0 CONT
MOVL C414 V=50.0 CONT
MOVL C415 V=50.0 CONT
MOVL C416 V=50.0 CONT
MOVL C417 V=50.0 CONT
MOVL C418 V=50.0 CONT
MOVL C419 V=50.0 CONT
MOVL C420 V=50.0 CONT
MOVL C421 V=50.0 CONT
MOVL C422 V=50.0 CONT
MOVL C423 V=50.0 CONT
MOVL C424 V=50.0 CONT
MOVL C425 V=50.0 CONT
MOVL C426 V=50.0 CONT
MOVL C427 V=50.0 CONT
MOVL C428 V=200.0 CONT
MOVL C429 V=200.0 CONT
MOVL C430 V=50.0 CONT
MOVL C431 V=50.0 CONT
MOVL C432 V=50.0 CONT
MOVL C433 V=50.0 CONT
MOVL C434 V=50.0 CONT
MOVL C435 V=50.0 CONT
MOVL C436 V=50.0 CONT
MOVL C437 V=50.0 CONT
MOVL C438 V=200.0 CONT
MOVL C439 V=200.0 CONT
MOVL C440 V=50.0 CONT
MOVL C441 V=50.0 CONT
MOVL C442 V=50.0 CONT
MOVL C443 V=50.0 CONT
MOVL C444 V=50.0 CONT
MOVL C445 V=50.0 CONT
MOVL C446 V=50.0 CONT
MOVL C447 V=50.0 CONT
MOVL C448 V=50.0 CONT
MOVL C449 V=50.0 CONT
MOVL C450 V=50.0 CONT
MOVL C451 V=50.0 CONT
MOVL C452 V=200.0 CONT
MOVL C453 V=200.0 CONT
MOVL C454 V=50.0 CONT
MOVL C455 V=50.0 CONT
MOVL C456 V=50.0 CONT
MOVL C457 V=50.0 CONT
MOVL C458 V=50.0 CONT
MOVL C459 V=50.0 CONT
MOVL C460 V=50.0 CONT
MOVL C461 V=50.0 CONT
MOVL C462 V=50.0 CONT
MOVL C463 V=50.0 CONT
MOVL C464 V=50.0 CONT
MOVL C465 V=50.0 CONT
MOVL C466 V=200.0 CONT
MOVL C467 V=200.0 CONT
MOVL C468 V=50.0 CONT
MOVL C469 V=50.0 CONT
MOVL C470 V=50.0 CONT
MOVL C471 V=50.0 CONT
MOVL C472 V=50.0 CONT
MOVL C473 V=50.0 CONT
MOVL C474 V=50.0 CONT
MOVL C475 V=50.0 CONT
MOVL C476 V=200.0 CONT
MOVL C477 V=200.0 CONT
MOVL C478 V=50.0 CONT
MOVL C479 V=50.0 CONT
MOVL C480 V=50.0 CONT
MOVL C481 V=50.0 CONT
MOVL C482 V=50.0 CONT
MOVL C483 V=50.0 CONT
MOVL C484 V=50.0 CONT
MOVL C485 V=50.0 CONT
MOVL C486 V=200.0 CONT
MOVL C487 V=200.0 CONT
MOVL C488 V=50.0 CONT
MOVL C489 V=50.0 CONT
MOVL C490 V=50.0 CONT
MOVL C491 V=50.0 CONT
MOVL C492 V=50.0 CONT
MOVL C493 V=50.0 CONT
MOVL C494 V=50.0 CONT
MOVL C495 V=50.0 CONT
MOVL C496 V=200.0 CONT
MOVL C497 V=200.0 CONT
MOVL C498 V=50.0 CONT
MOVL C499 V=50.0 CONT
MOVL C500 V=50.0 CONT
MOVL C501 V=50.0 CONT
MOVL C502 V=200.0 CONT
JUMP *1
END
